Staubli VAL3: onF8Event.pgx

program onF8Event()
  local string l_sItem
begin
  // look if the bButton is enable
  if bButton[7]
    //
    call loadPage("Disk://trajectory/TRACK/page_viewTrack",l_sItem)
    logMsg("[KERNEL] INTERFACE:PAGE Advance")
  endIf
end
